// TIA Portal V17 export
// export: Created 2024-10-17T14:16:16.6230221Z, ExportSetting WithDefaults, DisplayName Totally Integrated Automation Portal, DisplayVersion V17 Update 4, DisplayName TIA Portal Openness, DisplayVersion V17 Update 4, DisplayName TIA Portal Version Control Interface, DisplayVersion V17, DisplayName SINAMICS Startdrive Advanced, DisplayVersion V17 Update2, DisplayName SINAMICS Startdrive G130, G150, S120, S150, SINAMICS MV, S210, DisplayVersion V17 Update2, DisplayName SINAMICS Startdrive G110M, G120, G120C, G120D, G120P, G115D, DisplayVersion V17 Update2, DisplayName STEP 7 Professional, DisplayVersion V17 Update 4, DisplayName STEP 7 Safety, DisplayVersion V17, DisplayName WinCC Advanced / Unified PC, DisplayVersion V17 Update 4
TYPE "LPMLV2022_typeDiagnosticsEntry"
TITLE = LPMLV2022_typeDiagnosticsEntry
// Support: tech.team.motioncontrol@siemens.com
// stored: IsFailsafeCompliant false
   STRUCT
      timestamp { ExternalWritable := 'False'} : DTL;   // Timestamp for this entry
      UnitModeCurrent { ExternalWritable := 'False'} : SInt;   // Current unit mode
      StateCurrent { ExternalWritable := 'False'} : SInt;   // Current state
      UnitMode { ExternalWritable := 'False'} : SInt;   // Requested unit mode
      CntrlCmd { ExternalWritable := 'False'} : SInt;   // Request control command
      SC { ExternalWritable := 'False'} : Bool;   // State complete signal
      message { ExternalWritable := 'False'} : Byte;   // Message for this entry
   END_STRUCT;
END_TYPE
